PROGRAM PG_Consumer
VAR
	i:UDINT;
	k:UDINT;
END_VAR


//NovRam to File
FOR i:= 0 TO GVL.NovRamBufferRatio-1 DO
	GVL.fbNovRamToFileRingBuffer[i](udiNovRamIndex:=i);
END_FOR

//File to DB
FOR i:=0 TO gvl.NovRamBufferRatio-1 DO
	FOR k:=0 TO GVL.FileRingBufferRatio-1 DO
		gvl.fbFileRingBufferToDB[i][k](udiNovRam_BufferIndex:=i,udiFile_Index:=k);
	END_FOR
END_FOR

END_PROGRAM

(* stored: Version 1.1.0.1, ProductVersion 3.1.4024.11
   POU PG_Consumer: Id {62c174cb-6994-498a-a2d1-50bf0c0b0a87}, SpecialFunc None *)
